FUNCTION_BLOCK EventHelper EXTENDS FB_BaseFb
VAR_INPUT
//	pFlowID: 	POINTER TO DINT;
	pEvHeader: 	POINTER TO EventHeader_Typ;
	pEvPar: 	POINTER TO EventParam_Typ;
	Busy:BOOL:=FALSE;
	Done:BOOL;
END_VAR
VAR_OUTPUT
	
END_VAR
VAR
	EventReport :EventReport_Typ;
	InitDone:	 BOOL;
END_VAR

IF NOT InitDone THEN
	mInit();
	InitDone:= TRUE;
END_IF

METHOD mInit : BOOL
VAR_INPUT
END_VAR
SetLoggerCategoryName('Events');
END_METHOD

END_FUNCTION_BLOCK

(* stored: Version 1.1.0.1, ProductVersion 3.1.4024.3
   POU EventHelper: Id {20fd65cf-c883-0d8b-19ed-43645b78b546}, SpecialFunc None
   Method mInit: Id {26fd8f59-d260-44eb-9441-1f0c2395e49a} *)
